// Mitsubishi GX Works2 project: Exercicio sobre M W D   PLC: Q03UDV

PROGRAM MAIN
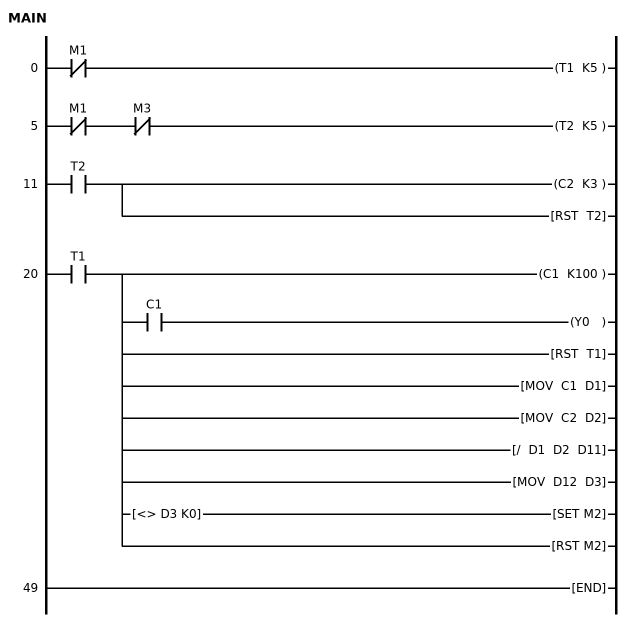
0     LDI     M1
      OUT     T1 K5
5     LDI     M1
      ANI     M3
      OUT     T2 K5
11    LD      T2
      OUT     C2 K3
      RST     T2
20    LD      T1
      OUT     C1 K100
      MPS
      AND     C1
      OUT     Y0
      MPP
      RST     T1
      MOV     C1 D1
      MOV     C2 D2
      /       D1 D2 D11
      MOV     D12 D3
      MPS
      AND<>   D3 K0
      SET     M2
      MPP
      RST     M2
49    END
END_PROGRAM
